Staubli VAL3: setSizeList.pgx

public program setSizeList(num nPx, num nPy, num nPBottomX, num nPBottomY)
begin
  nTopX=nTopX[1]=nPx
  nTopY=nPy
  nBottomX=nBottomX[1]=nPBottomX
  nBottomY=nPBottomY
end
